  ###################################################################################
  #
  # PATH GENERATOR 6 POINTS CURVE BUILT WITH 2 POINTS
  #
  ###################################################################################

  def execute_half_pipe(pose_1, pose_2,pose_transformation_air_nozzle_to_actual_tcp, depth, length_distance, width, angle, speed, spacing, address, output_type, blow_off_mode, passes):
    path_gen_poses = get_path_generator_6_points_poses(pose_1, pose_2, pose_transformation_air_nozzle_to_actual_tcp, depth, length_distance, width, angle)
    start_pose = p[path_gen_poses[0,0],path_gen_poses[0,1],path_gen_poses[0,2],path_gen_poses[0,3],path_gen_poses[0,4],path_gen_poses[0,5]]
    path_generator_node_id = setup_path_generator_6_points(path_gen_poses, speed, spacing)
    execute_path_generator_6_points(path_generator_node_id, start_pose,  address, output_type, blow_off_mode, passes)
  end

  def get_path_generator_6_points_poses(pose_2, pose_5,pose_transformation_air_nozzle_to_actual_tcp, depth=0.01, length=0, width=0.05, angle_deg=0):

    def offset_pose(pose, offset, offset_reference_frame, pose_transformation_air_nozzle_to_actual_tcp):
      pose_relative_to_ref_frame = express_pose_A_relative_to_pose_B(pose, offset_reference_frame)
      ref_frame_with_offset = pose_trans(offset_reference_frame, offset)
      pose_with_offset = pose_trans(ref_frame_with_offset, pose_relative_to_ref_frame)
      pose_with_offset_for_actual_tcp = pose_trans(pose_with_offset, pose_transformation_air_nozzle_to_actual_tcp)
      return pose_to_list(pose_with_offset_for_actual_tcp)
    end

    if(length > 0):
      middle_pose = interpolate_pose(pose_2, pose_5, 0.5)

      poses = get_symmetric_poses_from_middle(pose_2, pose_5, middle_pose, length)
      pose_2 = poses[0]
      pose_5 = poses[1]
    end

    path_ref_frame = list_to_pose(kinematics_rpc_server.reorientP1WithXTowardP2andZApproxP1Z(pose_2, pose_5))

    offset1 = pose_add(p[0,0,0,0,d2r(angle_deg),0], p[0, width,-depth,-d2r(angle_deg),0,0])
    offset2 = pose_add(p[0,0,0,0,d2r(angle_deg),0], p[0,     0,     0,              0,0,0])
    offset3 = pose_add(p[0,0,0,0,d2r(angle_deg),0], p[0,-width,-depth, d2r(angle_deg),0,0])

    pose_1_array = offset_pose(pose_2, offset1, path_ref_frame, pose_transformation_air_nozzle_to_actual_tcp)
    pose_2_array = offset_pose(pose_2, offset2, path_ref_frame, pose_transformation_air_nozzle_to_actual_tcp)
    pose_3_array = offset_pose(pose_2, offset3, path_ref_frame, pose_transformation_air_nozzle_to_actual_tcp)

    pose_4_array = offset_pose(pose_5, offset1, path_ref_frame, pose_transformation_air_nozzle_to_actual_tcp)
    pose_5_array = offset_pose(pose_5, offset2, path_ref_frame, pose_transformation_air_nozzle_to_actual_tcp)
    pose_6_array = offset_pose(pose_5, offset3, path_ref_frame, pose_transformation_air_nozzle_to_actual_tcp)

    return [pose_1_array, pose_2_array, pose_3_array, pose_4_array, pose_5_array, pose_6_array]
  end

  def setup_path_generator_6_points(pose_list, tcp_speed=0.1, spacing=0.02):

    def json_path_generator_node(pose_list, tcp_speed, spacing):

      SIX_POINTS_CURVE = 3
      OFFSET_TYPE_NONE = 0
      FORCE_OPPOSITE_SIDE = 2

      json = "{"
      json = concat(json, key_val("tcpSpeed", tcp_speed), ",")
      json = concat(json, key_val("poses", pose_list), ",")
      json = concat(json, key_val("avoidAbruptEnd", "false"), ",")
      json = concat(json, key_val("isSurfaceFillOn", "true"), ",")
      json = concat(json, key_val("spacing", spacing), ",")
      json = concat(json, key_val("pathType", SIX_POINTS_CURVE), ",")
      json = concat(json, key_val("offsetType",OFFSET_TYPE_NONE), ",")
      json = concat(json, key_val("endingMode", FORCE_OPPOSITE_SIDE), "}")

      return json
    end

    rq_path_generator_parent_id = 0
    path_generator_node_id = node_rpc_server.createPathGeneratorNode()
    node_rpc_server.fromjson(path_generator_node_id, json_path_generator_node(pose_list, tcp_speed, spacing))
    node_rpc_server.setparentid(path_generator_node_id, rq_path_generator_parent_id)

    return path_generator_node_id
  end

  def execute_path_generator_6_points(path_generator_node_id, pose_1, address = INVALID_OUTPUT_ADDRESS, output_type = MODBUS_TYPE, blow_off_mode = BLOW_OFF_MODE_NO_AIR, passes = 1):
    index = 0
    while (index < passes):
      movej(get_inverse_kin(pose_1))
      set_cleaning_digital_output(address, True, blow_off_mode, output_type)
      reset_node_executor()
      node_execution_thread = execute_node(path_generator_node_id, True)
      rq_continue_node_execution = False
      set_cleaning_digital_output(address, False, blow_off_mode, output_type)
      join node_execution_thread
      index = index + 1
    end
    node_rpc_server.deletenode(path_generator_node_id)
  end

  ###################################################################################
  #
  # Straight line trajectory
  #
  ###################################################################################

  def execute_straight_line(p1, p2,pose_transformation_air_nozzle_to_actual_tcp, accel=1.2, speed=0.25, distance = 0, angles = [0, 0, 0], address = INVALID_OUTPUT_ADDRESS, output_type = MODBUS_TYPE, blow_off_mode = BLOW_OFF_MODE_NO_AIR, passes = 1):
    offset_for_angles = p[0, 0, 0, d2r(angles[0]), d2r(angles[1]), d2r(angles[2])]
    p1 = pose_trans(p1, offset_for_angles)
    p2 = pose_trans(p2, offset_for_angles)

    # apply transformation to take into account that the actual tcp offset is not the same as the one that was used when the waypoints were saved:
    p1 = pose_trans(p1, pose_transformation_air_nozzle_to_actual_tcp)
    p2 = pose_trans(p2, pose_transformation_air_nozzle_to_actual_tcp)
    global air_output_adress = address

    qActual = get_actual_joint_positions()
    CleanPathId = node_rpc_server.createnewcleaningpathnode(p1, p2, qActual, passes, distance, accel, speed, blow_off_mode)

    reset_node_executor()
    if output_type == MODBUS_TYPE:
      air_thread = run modbusAirControlThread()
    elif output_type == STANDARD_TYPE:
      air_thread = run standardAirControlThread()
    end

    node_execution_thread = execute_node(CleanPathId, True)
    rq_continue_node_execution = False

    join node_execution_thread
    node_rpc_server.deletenode(CleanPathId)
    if output_type == MODBUS_TYPE or output_type == STANDARD_TYPE :
      kill air_thread
    end
  end

  ###################################################################################
  #
  # Cross trajectory
  #
  ###################################################################################

  def find_cross_trajectory_poses(p1, p2, height=0, width=0, p1_angles = [0, 0, 0], p2_angles = [0, 0, 0], p3_angles = [0, 0, 0], p4_angles = [0, 0, 0]):
    def find_side_poses(p0, p1):
      def find_side_pose(p0,p1,angle):
        p1_T_p0 = pose_trans(pose_inv(p0), p1)
        rotated_p0_by_90_degrees = pose_trans(p0, p[0, 0, 0, 0, 0, d2r(angle)])

        side_pose = pose_trans(rotated_p0_by_90_degrees, p1_T_p0)
        side_pose[3] = p0[3]
        side_pose[4] = p0[4]
        side_pose[5] = p0[5]

        return side_pose
      end

      p3= find_side_pose(p0, p1, 90)
      p4 = find_side_pose(p0, p1, 270)

      return [p3, p4]
    end

    def get_start_and_end_poses_based_on_distance(p1, p2, middle_pose, distance):
      if(distance == 0):
        start_pose = p1
        end_pose = p2
      else:
        poses = get_symmetric_poses_from_middle(p1, p2, middle_pose, distance)
        start_pose = poses[0]
        end_pose = poses[1]
      end
      return [start_pose, end_pose]
    end

    def get_side_poses_based_on_distance(p1, p2, middle_pose, width):
      if(width == 0):
        side_poses = find_side_poses(middle_pose, p1)
      else:
        poses = get_symmetric_poses_from_middle(p1, p2, middle_pose, width)
        side_poses = find_side_poses(middle_pose, poses[0])
      end

      return side_poses
    end

    def get_angle_offset(angles):
      return  p[0, 0, 0, d2r(angles[0]), d2r(angles[1]), d2r(angles[2])]
    end

    middle_pose = interpolate_pose(p1, p2, 0.5)

    start_and_end_poses = get_start_and_end_poses_based_on_distance(p1, p2, middle_pose, height)
    side_poses = get_side_poses_based_on_distance(p1, p2, middle_pose, width)

    p1_offset = get_angle_offset(p1_angles)
    p2_offset = get_angle_offset(p2_angles)
    p3_offset = get_angle_offset(p3_angles)
    p4_offset = get_angle_offset(p4_angles)

    start_and_end_poses[0] = pose_trans(start_and_end_poses[0], p1_offset)
    start_and_end_poses[1] = pose_trans(start_and_end_poses[1], p2_offset)
    side_poses[0] = pose_trans(side_poses[0], p3_offset)
    side_poses[1] = pose_trans(side_poses[1], p4_offset)

    return [middle_pose, start_and_end_poses[0], start_and_end_poses[1], side_poses[0], side_poses[1]]
  end

  def execute_cross_trajectory(p1, p2,pose_transformation_air_nozzle_to_actual_tcp, height=0, width=0, p1_angles = [0, 0, 0], p2_angles = [0, 0, 0], p3_angles = [0, 0, 0], p4_angles = [0, 0, 0], accel=1.2, speed=0.25,  address = INVALID_OUTPUT_ADDRESS, output_type = MODBUS_TYPE, blow_off_mode = BLOW_OFF_MODE_NO_AIR, passes = 1):

    cross_poses = find_cross_trajectory_poses(p1, p2, height, width, p1_angles, p2_angles, p3_angles, p4_angles)

    p0 = pose_trans(cross_poses[0], pose_transformation_air_nozzle_to_actual_tcp)
    p1 = pose_trans(cross_poses[1], pose_transformation_air_nozzle_to_actual_tcp)
    p2 = pose_trans(cross_poses[2], pose_transformation_air_nozzle_to_actual_tcp)
    p3 = pose_trans(cross_poses[3], pose_transformation_air_nozzle_to_actual_tcp)
    p4 = pose_trans(cross_poses[4], pose_transformation_air_nozzle_to_actual_tcp)

   index = 0

   while (index < passes):
     movej(get_inverse_kin(p0))
     set_cleaning_digital_output(address, True, blow_off_mode, output_type)
     movel(p1, accel, speed)
     movel(p2, accel, speed)
     movel(p0, accel, speed)
     movel(p3, accel, speed)
     movel(p4, accel, speed)
     set_cleaning_digital_output(address, False, blow_off_mode, output_type)
     index = index + 1
   end
  end

  def execute_waypoint_cross_trajectory(starting_pose, finishing_pose, accel=1.2, speed=0.25):
   movej(get_inverse_kin(starting_pose))
   movel(finishing_pose, accel, speed)
  end

  ###################################################################################
  #
  # Fermat spiral trajectory
  #
  ###################################################################################

  def execute_fermat_spiral(start_pose, end_pose,pose_transformation_air_nozzle_to_actual_tcp, max_radius = 0, angle = 0, number_of_turns = 1, speed = 0.25,address = INVALID_OUTPUT_ADDRESS, output_type = MODBUS_TYPE, blow_off_mode = BLOW_OFF_MODE_NO_AIR, passes = 1):
    def find_middle(start_pose, end_pose):
      alpha = 0.5
      return interpolate_pose(start_pose, end_pose, alpha)
    end

    def find_next_theta(spiral_constant, theta, speed):
      denom = spiral_constant * sqrt(1/(4*theta) + theta)
      theta_dot = speed / denom
      theta = theta + theta_dot * rq_controller_time_step
      return theta
    end

    def find_spiral_pose(theta, spiral_plane, center_pose, angle, spiral_constant, pose_transformation_air_nozzle_to_actual_tcp):
      local r = spiral_constant * sqrt(theta)
      local x = r * cos(theta)
      local y = r * sin(theta)

      local p2 = pose_trans(spiral_plane, p[x,y,0,0,0,0])
      local p3 = p[p2[0], p2[1], p2[2], center_pose[3], center_pose[4], center_pose[5]]
      local p4 = pose_trans(p3, pose_transformation_air_nozzle_to_actual_tcp)
      local p5 = pose_trans(p4, p[0, 0, 0, -d2r(angle)*cos(theta), -d2r(angle)*sin(theta), 0])
      return p5
    end

    def execute_outer_to_inner_spiral(start_pose, middle_pose, spiral_plane, pose_transformation_air_nozzle_to_actual_tcp, max_angle, angle, spiral_constant_nominal, speed, address, output_type, blow_off_mode):
      local theta = max_angle
      local max_r = point_dist(start_pose, middle_pose)
      local spiral_constant = -1 * spiral_constant_nominal
      local r = max_r
      local is_first_pose = True

      while (norm((r)) <= max_r):
        theta = find_next_theta(spiral_constant, theta, speed)
        if(theta < 0):
          break
        end

        r = spiral_constant * sqrt(theta)
        next_pose = find_spiral_pose(theta, spiral_plane, middle_pose, angle, spiral_constant, pose_transformation_air_nozzle_to_actual_tcp)

        if (is_first_pose):
          movej(get_inverse_kin(next_pose))
          set_cleaning_digital_output(address, True, blow_off_mode, output_type)
          is_first_pose = False
        else:
          servoj(get_inverse_kin(next_pose), t = rq_controller_time_step)
        end
      end
    end

    def execute_inner_to_outer_spiral(start_pose, middle_pose, spiral_plane, pose_transformation_air_nozzle_to_actual_tcp, angle, spiral_constant, speed):
      local theta = 0.0001
      local max_r = point_dist(start_pose, middle_pose)
      local r = 0

      while (norm(r) <= max_r):
        theta = find_next_theta(spiral_constant, theta, speed)
        r = spiral_constant * sqrt(theta)
        next_pose = find_spiral_pose(theta, spiral_plane, middle_pose, angle, spiral_constant, pose_transformation_air_nozzle_to_actual_tcp)
        servoj(get_inverse_kin(next_pose), t = rq_controller_time_step)
      end
    end

    max_angle = d2r(number_of_turns * 360)
    middle_pose = find_middle(start_pose, end_pose)

    if(max_radius > 0):
      poses = get_symmetric_poses_from_middle(start_pose, end_pose, middle_pose, max_radius * 2)
      start_pose = poses[0]
      end_pose = poses[1]
    end

    SPIRAL_CONSTANT = (point_dist(middle_pose, start_pose)) / sqrt(max_angle)

    spiral_plane = list_to_pose(kinematics_rpc_server.reorientP1WithXTowardP2andZApproxP1Z(middle_pose, end_pose))


    index = 0
    while(index < passes):
      execute_outer_to_inner_spiral(start_pose, middle_pose, spiral_plane,pose_transformation_air_nozzle_to_actual_tcp, max_angle, angle, SPIRAL_CONSTANT, speed, address, output_type, blow_off_mode)
      execute_inner_to_outer_spiral(end_pose, middle_pose, spiral_plane, pose_transformation_air_nozzle_to_actual_tcp, angle, SPIRAL_CONSTANT, speed)
      set_cleaning_digital_output(address, False, blow_off_mode, output_type)
      index = index + 1
    end
  end

  ###################################################################################
  #
  # ROBOTIQ VISE INSERTION
  #
  # - The first touch is performed in the direction of the gravity, regardless of
  #   the robot mounting orientation, tcp offset and TCP orientation
  # - Optional 2e et 3e touch are performed relative to TCP. They require that, at
  #   the moment that the insertion is performed, the TCP is oriented such that one
  #   axis is aligned with the gravity. The TCP axes for the 2e and 3e touch are
  #   chosen as the ones not aligned with the gravity.
  ###################################################################################
  def insert_in_vise(start_pose, end_pose, number_of_touch=3, forces=[10, 20, 20], invert_axis=False, move_to_end_pose=False):

    def list_by_scalar_multiply_(l1, scalar):
      result = l1
      i=0
      while i<length(result):
        result[i]=l1[i]*scalar
        i=i+1
      end
      return result
    end

    def find_gravity_direction(acceleration_direction, threshold):
      result = [False, False, False]
      i = 0
      while i < length(result):
        result[i] =  norm(acceleration_direction[i]) > threshold
        i = i + 1
      end
      return result
    end

    def get_axis(index, direction):
      axis = "XYZ"
      if direction < 0:
        sign = "-"
      elif direction > 0:
        sign = "+"
      else:
        popup("insert_in_vise:get_axis >>> direction cannot be 0. Fix it.")
        halt
      end
      return str_cat(str_sub(axis, index, 1), sign)
    end

    def direction_to_index(str):
      if "X" == str_sub(str, 0, 1):
        return 0
      elif "Y" == str_sub(str, 0, 1):
        return 1
      elif "Z" == str_sub(str, 0, 1):
        return 2
      else:
        popup("invalid direction :", str)
        halt
      end
    end

    def find_touch_direction(mask, direction):
      i = 0
      result = [0, 0, 0]
      while i < 3:
        if mask[i]:
          result[i] = direction[i]
        end
        i = i + 1
      end
      return result
    end

    def find_touch_direction_str(mask, direction):
      i = 0
      result = ""
      while i < 3:
        if mask[i]:
          result = str_cat(result, get_axis(i, direction[i]))
        end
        i = i + 1
      end
      return result
    end

    def invert(list):
      result = list
      i = 0
      while i < length(list):
        result[i] = not list[i]
        i = i + 1
      end
      return result
    end

    def assert_that_the_first_touch_is_aligned_with_an_axis(first_touch_direction_mask):
      i = 0
      counter = 0
      while i < length(first_touch_direction_mask):
        if first_touch_direction_mask[i]:
          counter = counter + 1
        end
        i = i + 1
      end

      if counter != 1:
        popup("One of the TCP axes must be perpendicular to the floor while loading the part in the vise.")
        halt
      end
    end

    def setup_nodes(forces, number_of_touch, first_touch_direction_mask, direction, second_direction_str, third_direction_str):
      def max_deviation_from(forces, enabled_axis):
        i = 0
        deviation = [0, 0, 0, 0, 0, 0]
        while i < 3:
          if forces[i] > 0:
            deviation[i] = 10
          elif forces[i] ==  0:
            deviation[i] = 10
          end
          i = i + 1
        end
        while i < 6:
          if enabled_axis[i]:
            deviation[i] = 0.35
          end
          i = i + 1
        end
        return deviation
      end

      def min_deviation_from(forces, enabled_axis):
        i = 0
        deviation = [0, 0, 0, 0, 0, 0]
        while i < 3:
          if forces[i] < 0:
            deviation[i] = -10
          elif forces[i] ==  0:
            deviation[i] = -10
          end
          i = i + 1
        end
        while i < 6:
          if enabled_axis[i]:
            deviation[i] = -0.35
          end
          i = i + 1
        end
        return deviation
      end

      def stiffness_from(forces):
        i = 0
        stiffness = [0, 0, 0, 100, 100, 100]
        while i < length(forces):
          if norm(forces[i]) > 0:
            stiffness[i] = 100
          else:
            stiffness[i] = 85
          end
          i = i + 1
        end
        return stiffness
      end

      def compute_final_forces(forces, number_of_touch, first_touch_direction_mask, direction, second_direction_str, third_direction_str):
        final_forces = [0, 0, 0]
        if number_of_touch > 0:
          i = 0
          while i < length(first_touch_direction_mask):
            if first_touch_direction_mask[i]:
              break
            end
            i = i + 1
          end
          final_forces[i] = direction[i] * forces[i]
        end
        if number_of_touch > 1:
          i = direction_to_index(second_direction_str)
          final_forces[i] = direction[i] * forces[i]
        end
        if number_of_touch > 2:
          i = direction_to_index(third_direction_str)
          final_forces[i] = direction[i] * forces[i]
        end
        return final_forces
      end

      def compute_enabled_axis(first_touch_direction_mask):
        enabled_axis = [True, True, True, False, False, False]
        i = 0
        while i < length(first_touch_direction_mask):
          if first_touch_direction_mask[i]:
            break
          end
          i = i + 1
        end
        enabled_axis[i + 3] = True

        return enabled_axis
      end

      final_forces = compute_final_forces(forces, number_of_touch, first_touch_direction_mask, direction, second_direction_str, third_direction_str)
      enabled_axis = compute_enabled_axis(first_touch_direction_mask)

      force_node_id = rq_setup_machine_tending_force_node(1, [final_forces[0], final_forces[1], final_forces[2], 0, 0, 0], stiffness_from
      (final_forces), min_deviation_from(final_forces, enabled_axis), max_deviation_from(final_forces, enabled_axis), rq_bool_array_to_string(enabled_axis), "false")
      movej_node_id = node_rpc_server.createnewmovejnode()
      node_rpc_server.setparentid(movej_node_id, force_node_id)

      return [force_node_id, movej_node_id]
    end

    def average_tool_acceleration_reading(n_samples, delay):
      n = n_samples
      reading = [0, 0, 0]
      while n > 0:
        reading = reading + get_tool_accelerometer_reading()
        sleep(delay)
        n = n - 1
      end
      return reading/n_samples
    end

    def linear_search_toward_gravity(force):
      # maybe add a stopj here to prevent acceleration reading to be influenced by robot movement
      flange_accel = average_tool_acceleration_reading(10, 0.1) # measured accel is oriented in gravity oposite direction
      flange_accel_pose = p[-flange_accel[0], -flange_accel[1], -flange_accel[2], 0, 0,0]
      p1 = translate_to_origin(get_actual_tool_flange_pose())
      gravity_dir_in_base_frame = pose_trans(p1, flange_accel_pose)

      # Find pose with z axis pointing in gravity direction:
      ref_frame_pose = list_to_pose(kinematics_rpc_server.poseFromZaxis([gravity_dir_in_base_frame[0], gravity_dir_in_base_frame[1], gravity_dir_in_base_frame[2]]))
      speed = 0.01
      abs_max_distance = 0.05

      surface_found = rq_linear_search_custom_frame("Z+", force, speed, abs_max_distance, ref_frame_pose)
      return surface_found
    end

    #### Actual insert_in_vise method ####
    movel(start_pose)
    zero_ftsensor()

    # 1. Use accelerometer reading to find touches directions:
    ACCELERATION_THRESHOLD = 8
    flange_accel = average_tool_acceleration_reading(10, 0.1)
    tcp_accel = pose_trans(pose_inv(get_tcp_offset()), p[flange_accel[0], flange_accel[1], flange_accel[2], 0, 0, 0])
    first_touch_direction_mask = find_gravity_direction(tcp_accel, ACCELERATION_THRESHOLD)
    assert_that_the_first_touch_is_aligned_with_an_axis(first_touch_direction_mask)

    direction_transform = pose_trans(pose_inv(start_pose), end_pose)
    direction = [direction_transform[0], direction_transform[1], direction_transform[2]]
    direction_sign = [direction[0]/norm(direction[0]), direction[1]/norm(direction[1]), direction[2]/norm(direction[2])]

    touch_direction_str = find_touch_direction_str(invert(first_touch_direction_mask), direction_sign)
    touch_direction = find_touch_direction(invert(first_touch_direction_mask), direction_sign)

    if invert_axis:
      second_direction_str = str_sub(touch_direction_str, 0, 2)
      third_direction_str = str_sub(touch_direction_str, 2, 4)
    else:
      second_direction_str = str_sub(touch_direction_str, 2, 4)
      third_direction_str = str_sub(touch_direction_str, 0, 2)
    end

    end_pose_orientation = translate_to_origin(end_pose)

    # 2. Prepare nodes:
    rq_cnc_insertion_node_ids = setup_nodes(forces, number_of_touch, first_touch_direction_mask, direction_sign, second_direction_str, third_direction_str)
    feature_tool = 1

    # 3. Perform touches:
    if number_of_touch > 0:
      surface_found = linear_search_toward_gravity(forces[0])
      if not surface_found:
        textmsg("Insertion in vise: First contact has not been found")
        popup("First contact has not been found", title="Insertion in vise", blocking=True)
        return UNDEFINED_THREAD_ID
      end
    end
    if number_of_touch > 1:
      surface_found = rq_linear_search_urcap(second_direction_str, forces[1], 0.01, 0.05, feature_tool)
      if not surface_found:
        textmsg("Insertion in vise: Second contact has not been found")
        popup("Second contact has not been found", title="Insertion in vise", blocking=True)
        return UNDEFINED_THREAD_ID
      end
    end
    if number_of_touch > 2:
      surface_found = rq_linear_search_urcap(third_direction_str, forces[2], 0.01, 0.05, feature_tool)
      if not surface_found:
        textmsg("Insertion in vise: Third contact has not been found")
        popup("Third contact has not been found", title="Insertion in vise", blocking=True)
        return UNDEFINED_THREAD_ID
      end
    end

    # 4. Move to end position:
    if not move_to_end_pose:
      end_pose = get_actual_tcp_pose()
    end

    node_rpc_server.movejdefinewaypoint(rq_cnc_insertion_node_ids[1], get_actual_joint_positions(), 1.0, 1.0)
    reset_node_executor()
    active_and_reset_node(rq_cnc_insertion_node_ids[0])
    node_execution_thread = execute_node(rq_cnc_insertion_node_ids[1], True)
    node_rpc_server.movejdefinewaypoint(rq_cnc_insertion_node_ids[1], get_inverse_kin(end_pose), 1.0, 1.0)
    execute_node(rq_cnc_insertion_node_ids[1])
    sleep(1)
    return node_execution_thread
  end

  ###################################################################################
  # AIR OUTPUT CONTROL
  ###################################################################################
  thread modbusAirControlThread():
    while (True):
      rq_air_value = read_input_boolean_register(101)
      modbus_set_output_signal(air_output_adress, rq_air_value, False)
      sleep(rq_controller_time_step)
    end
  end

  thread standardAirControlThread():
    while (True):
      rq_air_value = read_input_boolean_register(101)
      set_digital_out(air_output_adress, rq_air_value)
      sleep(rq_controller_time_step)
    end
  end
  def rq_set_output(output_type, address, value):
    if output_type == "MODBUS":
      modbus_set_output_signal(address, value)
    elif output_type == "STANDARD":
      set_standard_digital_out(address, value)
    end
  end

  def rq_digital_output_action(action, output_type, address, time_on=1, time_off=0.5, delay_after=0):
    if action == "PUSH_AND_HOLD":
      rq_set_output(output_type, address, True)
    elif action == "PUSH":
      rq_set_output(output_type, address, True)
      sleep(time_on)
      rq_set_output(output_type, address, False)
    elif action == "DOUBLE_PUSH":
      rq_set_output(output_type, address, True)
      sleep(time_on)
      rq_set_output(output_type, address, False)
      sleep(time_off)
      rq_set_output(output_type, address, True)
      sleep(time_on)
      rq_set_output(output_type, address, False)
    elif action == "RELEASE":
      rq_set_output(output_type, address, False)
    end
    sleep(delay_after)
  end
  def json_kinematic_parameters_ratio(ratio):
    json = "{"
    json = concat(json, key_val("kinematicParametersRatio", ratio), "}")
    return json
  end

  def execute_move_along_trail(trail_node_id, joint_positions, kinematic_parameters_ratio):
    node_rpc_server.fromjson(trail_node_id, json_kinematic_parameters_ratio(kinematic_parameters_ratio))
    roadmap_state = node_rpc_server.initRoadmap(trail_node_id, joint_positions)
    path_time = roadmap_state[0]

    if(path_time > 0.0):
      reset_node_executor()
      node_execution_thread = execute_node(trail_node_id, True)
      kill node_execution_thread
    end
  end
    global servojId = 2
  rq_collision_detection_stop()
  # end: URCap Installation Node
  global Loop_1=0
  global Loop_2=0
  global P1=p[0,0,0,0,0,0]
  global P2=p[0,0,0,0,0,0]
  global P3=p[0,0,0,0,0,0]
  global P4=p[0,0,0,0,0,0]
  global Plate=p[0.0249751273065488,0.315444418995817,-0.002979446203698388,2.4062421505685623,-2.0195268274258926,2.0269178961854212E-4]
  global PlateSlot=p[0.300029473663405,0.21098389212496838,0.09999602225772891,-1.5172339309352096,0.4787574757529798,0.4782972175474087]
  global Push=p[0.30076538865744507,-0.3222894527764391,0.02802936275719442,0.9445418379537732,2.996231629718085,-3.1473923717280155E-4]
  global Rebar=p[0.18104878031330549,0.14999304691346624,0.007927916021551962,2.7864361304382914,1.4505933834983582,6.744682085333812E-5]
  global RebarSlot=p[0.2999891101196033,-0.050016493917625006,0.0600028647678886,2.786182363334521,1.4503518590317919,-2.993328738756438E-4]
  global o100=p[0,0,0.1,0,0,0]
  global o150=p[0,0,0.15,0,0,0]
  global o50=p[0,0,0.05,0,0,0]
  $ 2 "Robot Program"
  $ 3 "MoveJ"
  $ 4 "Rest" "breakAfter"
  movej(get_inverse_kin(p[.249974193900, .190010098788, .200047314165, -1.450629691050, 2.786568775509, -.000008157466], qnear=[-2.8488815466518975, -1.5533502737616, 1.7855463027947795, 1.3384930033544513, 1.563626050947951, -2.2383263746852737]), a=1.3962634015954636, v=1.0471975511965976)
  $ 5 "Loop 4 times"
  Loop_1 = 0
  while (Loop_1 < 4):
    $ 6 "'Pick plate'"
    # 'Pick plate'
    $ 7 "P1≔pose_add(Plate, o100)"
    global P1= pose_add (Plate, o100)
    $ 8 "P2≔pose_add(Plate, o50)"
    global P2= pose_add (Plate, o50)
    $ 9 "MoveJ"
    $ 10 "Above_plates" "breakAfter"
    movej(get_inverse_kin(p[.024945049144, .315448884679, .147023291383, 2.406351017142, -2.019349816061, .000241364861], qnear=[-2.003760639820306, -1.5083611647227189, 1.8802962303155475, 1.1990411961201044, 1.5637578964245151, -2.177393261586011]), a=1.3962634015954636, v=1.0471975511965976, r=0.01)
    $ 11 "MoveL"
    $ 13 "P2" "breakAfter"
    movel(pose_trans(p[0.0,0.0,0.0,0.0,0.0,0.0], P2), a=1.2, v=0.1)
    $ 14 "Set DO[2]=Off"
    set_standard_digital_out(2, False)
    $ 15 "Set DO[3]=On"
    set_standard_digital_out(3, True)
    $ 16 "Wait: 0.5"
    sleep(0.5)
    $ 17 "Set DO[3]=Off"
    set_standard_digital_out(3, False)
    $ 18 "Plate" "breakAfter"
    movel(pose_trans(p[0.0,0.0,0.0,0.0,0.0,0.0], Plate), a=1.2, v=0.1)
    $ 20 "P2" "breakAfter"
    movel(pose_trans(p[0.0,0.0,0.0,0.0,0.0,0.0], P2), a=1.2, v=0.1, r=0.01)
    $ 22 "MoveJ"
    $ 23 "Above_plates" "breakAfter"
    movej(get_inverse_kin(p[.024945049144, .315448884679, .147023291383, 2.406351017142, -2.019349816061, .000241364861], qnear=[-2.003760639820306, -1.5083611647227189, 1.8802962303155475, 1.1990411961201044, 1.5637578964245151, -2.177393261586011]), a=1.3962634015954636, v=1.0471975511965976, r=0.01)
    $ 24 "MoveL"
    $ 25 "RotatePlate" "breakAfter"
    movel(p[.149914523802, .336502068655, .356770919309, -1.538768807768, .524337562537, .526894930491], a=0.1, v=0.1)
    $ 26 "Plate≔pose_add(Plate, p[0,0,-0.003,0,0,0])"
    global Plate= pose_add (Plate, p[0,0,-0.003,0,0,0])
    $ 27 "'Drop plate'"
    # 'Drop plate'
    $ 28 "P1≔pose_add(PlateSlot,o150)"
    global P1=pose_add(PlateSlot,o150)
    $ 29 "P2≔pose_add(PlateSlot, o50)"
    global P2= pose_add (PlateSlot, o50)
    $ 30 "P3≔pose_add(PlateSlot, p[0,-0.025,0.025,0,0,0])"
    global P3= pose_add (PlateSlot, p[0,-0.025,0.025,0,0,0])
    $ 31 "P4≔pose_add(PlateSlot, p[0,-0.025,0.15,0,0,0])"
    global P4= pose_add (PlateSlot, p[0,-0.025,0.15,0,0,0])
    $ 32 "MoveJ"
    $ 33 "Above_plate_s" "breakAfter"
    movej(get_inverse_kin(p[.300721055666, .211018460361, .280007921139, -1.517276813467, .478662626415, .478315411592], qnear=[-3.5531768281373743, -1.7788722915284474, 2.115790250507308, -0.3209439244459755, -0.41066959272423365, -2.5479184221414872]), a=1.3962634015954636, v=1.0471975511965976, r=0.01)
    $ 34 "MoveL"
    $ 35 "P1" "breakAfter"
    movel(pose_trans(p[0.0,0.0,0.0,0.0,0.0,0.0], P1), a=1.2, v=0.1, r=0.01)
    $ 36 "P2" "breakAfter"
    movel(pose_trans(p[0.0,0.0,0.0,0.0,0.0,0.0], P2), a=1.2, v=0.05, r=0.01)
    $ 37 "PlateSlot" "breakAfter"
    movel(pose_trans(p[0.0,0.0,0.0,0.0,0.0,0.0], PlateSlot), a=1.2, v=0.05)
    $ 38 "Set DO[3]=Off"
    set_standard_digital_out(3, False)
    $ 39 "Set DO[2]=On"
    set_standard_digital_out(2, True)
    $ 40 "Wait: 0.5"
    sleep(0.5)
    $ 41 "Set DO[2]=Off"
    set_standard_digital_out(2, False)
    $ 42 "P3" "breakAfter"
    movel(pose_trans(p[0.0,0.0,0.0,0.0,0.0,0.0], P3), a=1.2, v=0.05)
    $ 43 "P4" "breakAfter"
    movel(pose_trans(p[0.0,0.0,0.0,0.0,0.0,0.0], P4), a=1.2, v=0.25, r=0.01)
    $ 44 "MoveJ"
    $ 45 "Above_plate_s" "breakAfter"
    movej(get_inverse_kin(p[.300721055666, .211018460361, .280007921139, -1.517276813467, .478662626415, .478315411592], qnear=[-3.5531768281373743, -1.7788722915284474, 2.115790250507308, -0.3209439244459755, -0.41066959272423365, -2.5479184221414872]), a=1.3962634015954636, v=1.0471975511965976, r=0.01)
    $ 46 "If Loop_1 % 2≠0"
    if (Loop_1 % 2 != 0):
      $ 47 "PlateSlot≔pose_add(PlateSlot, p[0.1,-0.006,0,0,0,0])"
      global PlateSlot= pose_add (PlateSlot, p[0.1,-0.006,0,0,0,0])
    else:
      $ 48 "Else" "noBreak"
      $ 49 "PlateSlot≔pose_add(PlateSlot, p[0.1,0.006,0,0,0,0])"
      global PlateSlot= pose_add (PlateSlot, p[0.1,0.006,0,0,0,0])
    end
    Loop_1 = Loop_1 + 1
  end
  $ 51 "Loop 4 times"
  Loop_2 = 0
  while (Loop_2 < 4):
    $ 52 "'Pick rebar'"
    # 'Pick rebar'
    $ 53 "P1≔pose_add(Rebar, o50)"
    global P1= pose_add (Rebar, o50)
    $ 54 "P2≔pose_add(Rebar, p[-0.01,0,0.025,0,0,0])"
    global P2= pose_add (Rebar, p[-0.01,0,0.025,0,0,0])
    $ 55 "P3≔pose_add(Rebar, p[-0.01,0,0.2,0,0,0])"
    global P3= pose_add (Rebar, p[-0.01,0,0.2,0,0,0])
    $ 56 "MoveJ"
    $ 57 "Above_rebar_s" "breakAfter"
    movej(get_inverse_kin(p[.300000000000, -.064983718114, .210025402337, 2.786231090849, 1.450518339391, -.000243746251], qnear=[-3.719007828494142, -2.0581159729885687, 2.1365851752907536, -1.6492773407251162, -1.5640363465239027, -3.1091725379446657]), a=1.3962634015954636, v=1.0471975511965976, r=0.01)
    $ 58 "MoveL"
    $ 59 "P1" "breakAfter"
    movel(pose_trans(p[0.0,0.0,0.0,0.0,0.0,0.0], P1), a=1.2, v=0.1)
    $ 60 "Set DO[2]=Off"
    set_standard_digital_out(2, False)
    $ 61 "Set DO[3]=On"
    set_standard_digital_out(3, True)
    $ 62 "Wait: 0.5"
    sleep(0.5)
    $ 63 "Set DO[3]=Off"
    set_standard_digital_out(3, False)
    $ 64 "Rebar" "breakAfter"
    movel(pose_trans(p[0.0,0.0,0.0,0.0,0.0,0.0], Rebar), a=1.2, v=0.1)
    $ 65 "P2" "breakAfter"
    movel(pose_trans(p[0.0,0.0,0.0,0.0,0.0,0.0], P2), a=1.2, v=0.1, r=0.01)
    $ 66 "P3" "breakAfter"
    movel(pose_trans(p[0.0,0.0,0.0,0.0,0.0,0.0], P3), a=1.2, v=0.1)
    $ 67 "MoveJ"
    $ 68 "Above_rebar_s" "breakAfter"
    movej(get_inverse_kin(p[.300000000000, -.064983718114, .210025402337, 2.786231090849, 1.450518339391, -.000243746251], qnear=[-3.719007828494142, -2.0581159729885687, 2.1365851752907536, -1.6492773407251162, -1.5640363465239027, -3.1091725379446657]), a=1.3962634015954636, v=1.0471975511965976, r=0.01)
    $ 69 "Rebar≔pose_add(Rebar, p[0.015,0,-0.005,0,0,0])"
    global Rebar= pose_add (Rebar, p[0.015,0,-0.005,0,0,0])
    $ 70 "'Drop rebar'"
    # 'Drop rebar'
    $ 71 "P1≔pose_add(RebarSlot, o50)"
    global P1= pose_add (RebarSlot, o50)
    $ 72 "P2≔pose_add(RebarSlot, o150)"
    global P2= pose_add (RebarSlot, o150)
    $ 73 "MoveJ"
    $ 74 "Above_rebar_s" "breakAfter"
    movej(get_inverse_kin(p[.300000000000, -.064983718114, .210025402337, 2.786231090849, 1.450518339391, -.000243746251], qnear=[-3.719007828494142, -2.0581159729885687, 2.1365851752907536, -1.6492773407251162, -1.5640363465239027, -3.1091725379446657]), a=1.3962634015954636, v=1.0471975511965976, r=0.01)
    $ 75 "MoveL"
    $ 76 "P1" "breakAfter"
    movel(pose_trans(p[0.0,0.0,0.0,0.0,0.0,0.0], P1), a=1.2, v=0.25, r=0.01)
    $ 77 "RebarSlot" "breakAfter"
    movel(pose_trans(p[0.0,0.0,0.0,0.0,0.0,0.0], RebarSlot), a=1.2, v=0.1)
    $ 78 "Set DO[3]=Off"
    set_standard_digital_out(3, False)
    $ 79 "Set DO[2]=On"
    set_standard_digital_out(2, True)
    $ 80 "Wait: 0.5"
    sleep(0.5)
    $ 81 "Set DO[2]=Off"
    set_standard_digital_out(2, False)
    $ 82 "P1" "breakAfter"
    movel(pose_trans(p[0.0,0.0,0.0,0.0,0.0,0.0], P1), a=1.2, v=0.25, r=0.01)
    $ 83 "MoveJ"
    $ 84 "P2" "breakAfter"
    movej(P2, a=1.3962634015954636, v=1.0471975511965976, r=0.01)
    $ 86 "RebarSlot≔pose_add(RebarSlot, p[0.1,0,0,0,0,0])"
    global RebarSlot= pose_add (RebarSlot, p[0.1,0,0,0,0,0])
    $ 87 "'Push'"
    # 'Push'
    $ 88 "P1≔pose_add(Push, p[0,-0.025,0,0,0,0])"
    global P1= pose_add (Push, p[0,-0.025,0,0,0,0])
    $ 89 "P2≔pose_add(Push, o50)"
    global P2= pose_add (Push, o50)
    $ 90 "P3≔pose_add(Push, p[0,0.05,0,0,0,0])"
    global P3= pose_add (Push, p[0,0.05,0,0,0,0])
    $ 91 "P4≔pose_add(Push, o150)"
    global P4= pose_add (Push, o150)
    $ 92 "MoveJ"
    $ 93 "P4" "breakAfter"
    movej(P4, a=1.3962634015954636, v=1.0471975511965976)
    $ 95 "MoveL"
    $ 96 "P1" "breakAfter"
    movel(pose_trans(p[0.0,0.0,0.0,0.0,0.0,0.0], P1), a=1.2, v=0.25, r=0.01)
    $ 97 "Push" "breakAfter"
    movel(pose_trans(p[0.0,0.0,0.0,0.0,0.0,0.0], Push), a=0.1, v=0.02)
    # begin: URCap Program Node
    #   Source: Robotiq_Copilot, 1.30.5.37741, Robotiq Inc.
    #   Type: Insertion
    $ 98 "Insertion"
    rq_ft_sensor_disconnected_check()
    # begin: URCap Program Node
    #   Source: Robotiq_Copilot, 1.30.5.37741, Robotiq Inc.
    #   Type: Zero FT Sensor
    $ 99 "Zero FT Sensor" "noBreak"
    rq_ft_sensor_disconnected_check()
    rq_wait_ft_sensor_steady(2000)
    rq_zero_sensor()
    # end: URCap Program Node
    # begin: URCap Program Node
    #   Source: Robotiq_Copilot, 1.30.5.37741, Robotiq Inc.
    #   Type: Linear
    $ 100 "Linear" "noBreak"
    rq_ft_sensor_disconnected_check()
    surface_found = rq_linear_search_urcap("Y+", 5.000, 0.010, 0.100, 0)
    # begin: URCap Program Node
    #   Source: Robotiq_Copilot, 1.30.5.37741, Robotiq Inc.
    #   Type: On error
    $ 101 "On error" "noBreak"
    if not(surface_found):
      $ 102 "'Correct'" "noBreak"
      # 'Correct'
    end
    # end: URCap Program Node
    # end: URCap Program Node
    # end: URCap Program Node
    $ 106 "P2" "breakAfter"
    movel(pose_trans(p[0.0,0.0,0.0,0.0,0.0,0.0], P2), a=1.2, v=0.25, r=0.01)
    $ 107 "MoveJ"
    $ 108 "Above_rebar_s" "breakAfter"
    movej(get_inverse_kin(p[.300000000000, -.064983718114, .210025402337, 2.786231090849, 1.450518339391, -.000243746251], qnear=[-3.719007828494142, -2.0581159729885687, 2.1365851752907536, -1.6492773407251162, -1.5640363465239027, -3.1091725379446657]), a=1.3962634015954636, v=1.0471975511965976)
    $ 110 "Push≔pose_add(Push, p[0.1,0,0,0,0,0])"
    global Push= pose_add (Push, p[0.1,0,0,0,0,0])
    Loop_2 = Loop_2 + 1
  end
  $ 111 "MoveJ"
  $ 112 "Rest" "breakAfter"
  movej(get_inverse_kin(p[.249974193900, .190010098788, .200047314165, -1.450629691050, 2.786568775509, -.000008157466], qnear=[-2.8488815466518975, -1.5533502737616, 1.7855463027947795, 1.3384930033544513, 1.563626050947951, -2.2383263746852737]), a=1.3962634015954636, v=1.0471975511965976)
end
